// TIA Portal V17 export
// export: Created 2024-01-30T08:49:11.8179475Z, ExportSetting WithDefaults, DisplayName Totally Integrated Automation Portal, DisplayVersion V17 Update 6, DisplayName TIA Portal Openness, DisplayVersion V17 Update 6, DisplayName TIA Portal Version Control Interface, DisplayVersion V17, DisplayName STEP 7 Professional, DisplayVersion V17 Update 6, DisplayName STEP 7 Safety, DisplayVersion V17 Update 6, DisplayName WinCC Advanced, DisplayVersion V17 Update 6
FUNCTION "FC_TransferDataPLC_LJX8000" : Void   // FC4, LAD
{ S7_Optimized_Access := 'TRUE' }
VERSION : 0.1
// stored: AutoNumber true, IsIECCheckEnabled false, SetENOAutomatically false, UDAEnableTagReadback false
BEGIN

REGION Network 1: PLC to LJ_X8000 bits
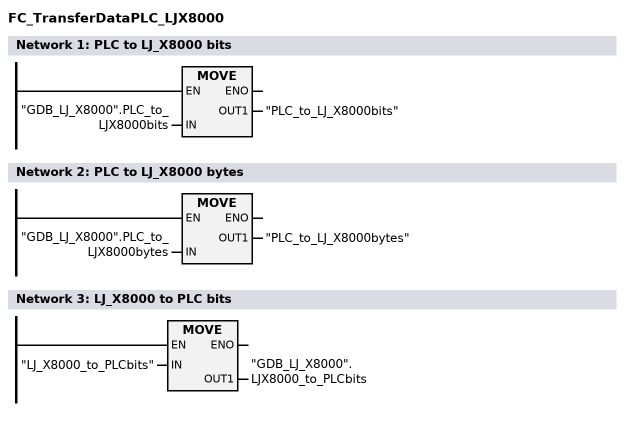
   RUNG wire#powerrail
      Move(in := "GDB_LJ_X8000".PLC_to_LJX8000bits, out1 => "PLC_to_LJ_X8000bits")
   END_RUNG
   // the same network as SCL:
   "PLC_to_LJ_X8000bits" := "GDB_LJ_X8000".PLC_to_LJX8000bits;
END_REGION

REGION Network 2: PLC to LJ_X8000 bytes
   RUNG wire#powerrail
      Move(in := "GDB_LJ_X8000".PLC_to_LJX8000bytes, out1 => "PLC_to_LJ_X8000bytes")
   END_RUNG
   // the same network as SCL:
   "PLC_to_LJ_X8000bytes" := "GDB_LJ_X8000".PLC_to_LJX8000bytes;
END_REGION

REGION Network 3: LJ_X8000 to PLC bits
   RUNG wire#powerrail
      Move(in := "LJ_X8000_to_PLCbits", out1 => "GDB_LJ_X8000".LJX8000_to_PLCbits)
   END_RUNG
   // the same network as SCL:
   "GDB_LJ_X8000".LJX8000_to_PLCbits := "LJ_X8000_to_PLCbits";
END_REGION
END_FUNCTION
